// Mitsubishi GX Works2 project: 2023-05-10 #1 생산자동화기능사 1번   PLC: Q03UDV
// 생산자동화기능사

// global labels: Global1
VAR_GLOBAL
  PB1 AT X0 : BOOL;
  PB2 AT X1 : BOOL;
  정지 AT X2 : BOOL;
  공급후진 AT X3 : BOOL;
  공급전진 AT X4 : BOOL;
  가공후진 AT X5 : BOOL;
  가공전진 AT X6 : BOOL;
  송출후진 AT X7 : BOOL;
  송출전진 AT X8 : BOOL;
  배출후진 AT X9 : BOOL;
  배출전진 AT X0A : BOOL;
  매거진 AT X0B : BOOL;
  금속센서 AT X0F : BOOL;
  PB3 AT X0C : BOOL;
  적색 AT Y20 : BOOL;
  황색 AT Y21 : BOOL;
  녹색 AT Y22 : BOOL;
  공급1 AT Y23 : BOOL;
  공급2 AT Y24 : BOOL;
  가공 AT Y25 : BOOL;
  드릴 AT Y26 : BOOL;
  송출 AT Y27 : BOOL;
  배출 AT Y28 : BOOL;
  컨베이어 AT Y29 : BOOL;
  METAL : INT;
END_VAR

PROGRAM 테스트동작
VAR
  STATE : INT;
END_VAR
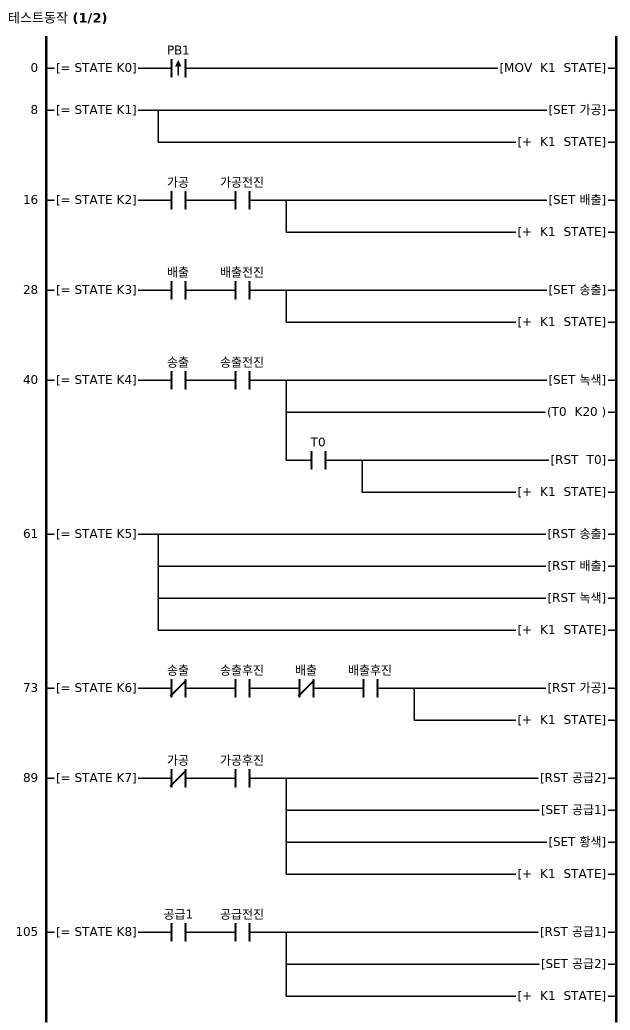
0     LD=     STATE K0
      ANDP    PB1
      MOV     K1 STATE
8     LD=     STATE K1
      SET     가공
      +       K1 STATE
16    LD=     STATE K2
      AND     가공
      AND     가공전진
      SET     배출
      +       K1 STATE
28    LD=     STATE K3
      AND     배출
      AND     배출전진
      SET     송출
      +       K1 STATE
40    LD=     STATE K4
      AND     송출
      AND     송출전진
      SET     녹색
      OUT     T0 K20
      AND     T0
      RST     T0
      +       K1 STATE
61    LD=     STATE K5
      RST     송출
      RST     배출
      RST     녹색
      +       K1 STATE
73    LD=     STATE K6
      ANI     송출
      AND     송출후진
      ANI     배출
      AND     배출후진
      RST     가공
      +       K1 STATE
89    LD=     STATE K7
      ANI     가공
      AND     가공후진
      RST     공급2
      SET     공급1
      SET     황색
      +       K1 STATE
105   LD=     STATE K8
      AND     공급1
      AND     공급전진
      RST     공급1
      SET     공급2
      +       K1 STATE
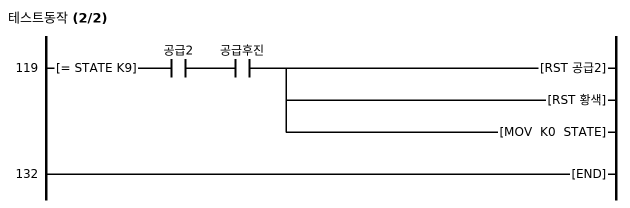
119   LD=     STATE K9
      AND     공급2
      AND     공급후진
      RST     공급2
      RST     황색
      MOV     K0 STATE
132   END
END_PROGRAM

PROGRAM 연속동작
VAR
  COUNT : INT;
  STATE : INT;
  RESET : INT;
END_VAR
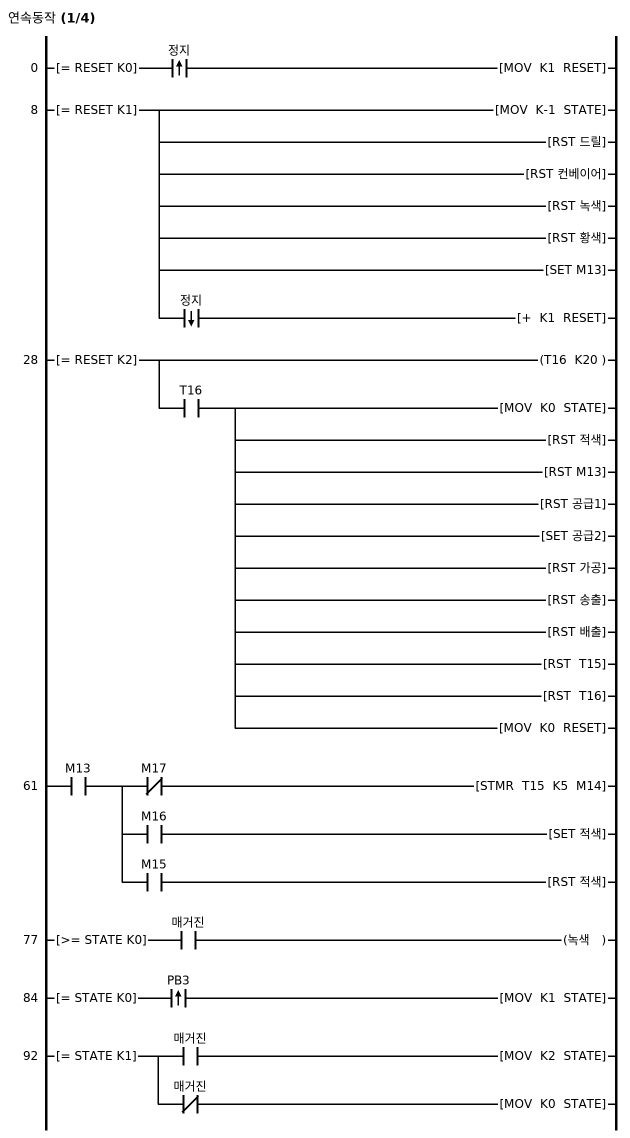
0     LD=     RESET K0
      ANDP    정지
      MOV     K1 RESET
8     LD=     RESET K1
      MOV     K-1 STATE
      RST     드릴
      RST     컨베이어
      RST     녹색
      RST     황색
      SET     M13
      ANDF    정지
      +       K1 RESET
28    LD=     RESET K2
      OUT     T16 K20
      AND     T16
      MOV     K0 STATE
      RST     적색
      RST     M13
      RST     공급1
      SET     공급2
      RST     가공
      RST     송출
      RST     배출
      RST     T15
      RST     T16
      MOV     K0 RESET
61    LD      M13
      MPS
      ANI     M17
      STMR    T15 K5 M14
      MRD
      AND     M16
      SET     적색
      MPP
      AND     M15
      RST     적색
77    LD>=    STATE K0
      AND     매거진
      OUT     녹색
84    LD=     STATE K0
      ANDP    PB3
      MOV     K1 STATE
92    LD=     STATE K1
      MPS
      AND     매거진
      MOV     K2 STATE
      MPP
      ANI     매거진
      MOV     K0 STATE
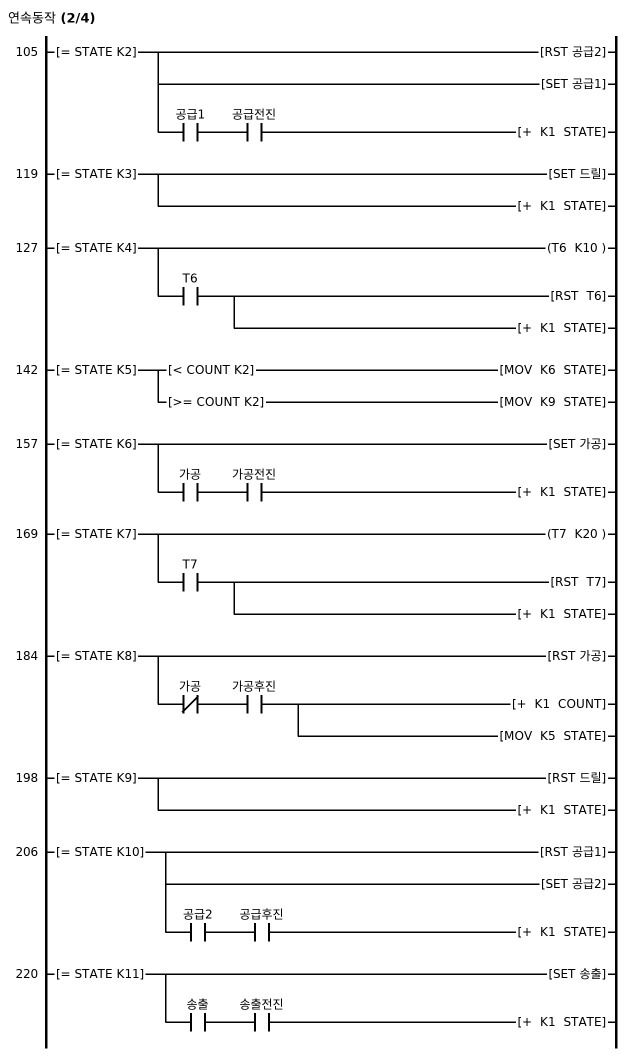
105   LD=     STATE K2
      RST     공급2
      SET     공급1
      AND     공급1
      AND     공급전진
      +       K1 STATE
119   LD=     STATE K3
      SET     드릴
      +       K1 STATE
127   LD=     STATE K4
      OUT     T6 K10
      AND     T6
      RST     T6
      +       K1 STATE
142   LD=     STATE K5
      MPS
      AND<    COUNT K2
      MOV     K6 STATE
      MPP
      AND>=   COUNT K2
      MOV     K9 STATE
157   LD=     STATE K6
      SET     가공
      AND     가공
      AND     가공전진
      +       K1 STATE
169   LD=     STATE K7
      OUT     T7 K20
      AND     T7
      RST     T7
      +       K1 STATE
184   LD=     STATE K8
      RST     가공
      ANI     가공
      AND     가공후진
      +       K1 COUNT
      MOV     K5 STATE
198   LD=     STATE K9
      RST     드릴
      +       K1 STATE
206   LD=     STATE K10
      RST     공급1
      SET     공급2
      AND     공급2
      AND     공급후진
      +       K1 STATE
220   LD=     STATE K11
      SET     송출
      AND     송출
      AND     송출전진
      +       K1 STATE
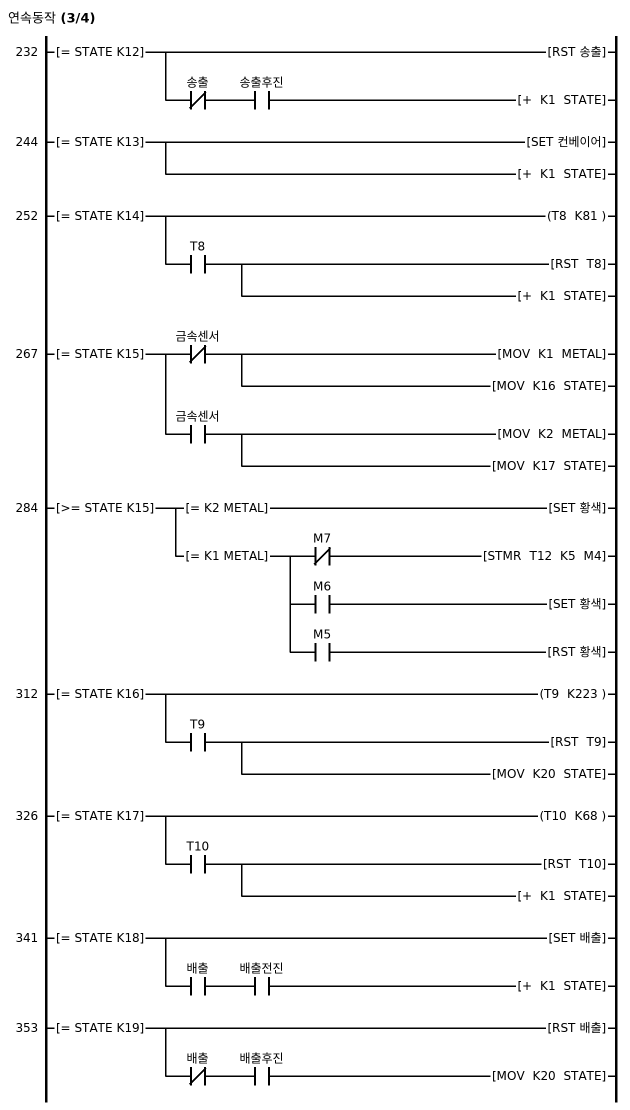
232   LD=     STATE K12
      RST     송출
      ANI     송출
      AND     송출후진
      +       K1 STATE
244   LD=     STATE K13
      SET     컨베이어
      +       K1 STATE
252   LD=     STATE K14
      OUT     T8 K81
      AND     T8
      RST     T8
      +       K1 STATE
267   LD=     STATE K15
      MPS
      ANI     금속센서
      MOV     K1 METAL
      MOV     K16 STATE
      MPP
      AND     금속센서
      MOV     K2 METAL
      MOV     K17 STATE
284   LD>=    STATE K15
      MPS
      AND=    K2 METAL
      SET     황색
      MPP
      AND=    K1 METAL
      MPS
      ANI     M7
      STMR    T12 K5 M4
      MRD
      AND     M6
      SET     황색
      MPP
      AND     M5
      RST     황색
312   LD=     STATE K16
      OUT     T9 K223
      AND     T9
      RST     T9
      MOV     K20 STATE
326   LD=     STATE K17
      OUT     T10 K68
      AND     T10
      RST     T10
      +       K1 STATE
341   LD=     STATE K18
      SET     배출
      AND     배출
      AND     배출전진
      +       K1 STATE
353   LD=     STATE K19
      RST     배출
      ANI     배출
      AND     배출후진
      MOV     K20 STATE
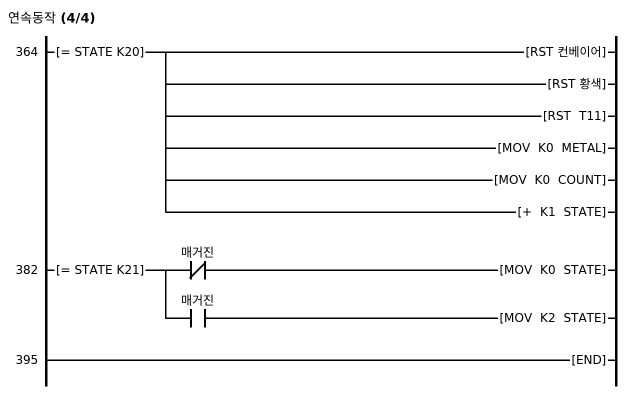
364   LD=     STATE K20
      RST     컨베이어
      RST     황색
      RST     T11
      MOV     K0 METAL
      MOV     K0 COUNT
      +       K1 STATE
382   LD=     STATE K21
      MPS
      ANI     매거진
      MOV     K0 STATE
      MPP
      AND     매거진
      MOV     K2 STATE
395   END
END_PROGRAM

PROGRAM 단속동작
VAR
  STATE : INT;
  RESET : INT;
END_VAR
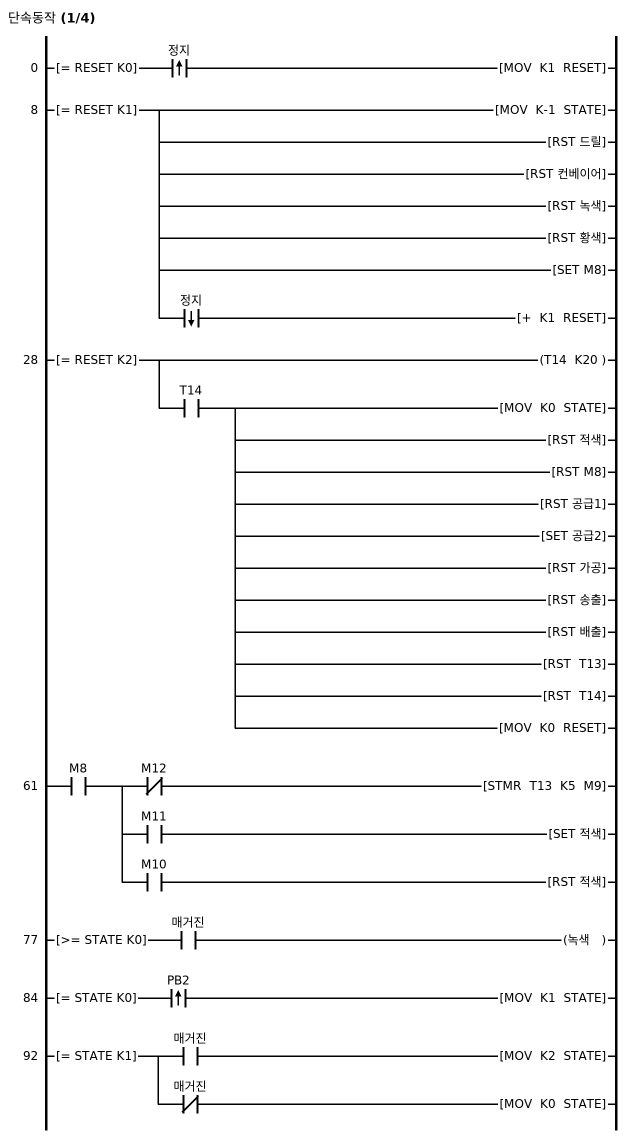
0     LD=     RESET K0
      ANDP    정지
      MOV     K1 RESET
8     LD=     RESET K1
      MOV     K-1 STATE
      RST     드릴
      RST     컨베이어
      RST     녹색
      RST     황색
      SET     M8
      ANDF    정지
      +       K1 RESET
28    LD=     RESET K2
      OUT     T14 K20
      AND     T14
      MOV     K0 STATE
      RST     적색
      RST     M8
      RST     공급1
      SET     공급2
      RST     가공
      RST     송출
      RST     배출
      RST     T13
      RST     T14
      MOV     K0 RESET
61    LD      M8
      MPS
      ANI     M12
      STMR    T13 K5 M9
      MRD
      AND     M11
      SET     적색
      MPP
      AND     M10
      RST     적색
77    LD>=    STATE K0
      AND     매거진
      OUT     녹색
84    LD=     STATE K0
      ANDP    PB2
      MOV     K1 STATE
92    LD=     STATE K1
      MPS
      AND     매거진
      MOV     K2 STATE
      MPP
      ANI     매거진
      MOV     K0 STATE
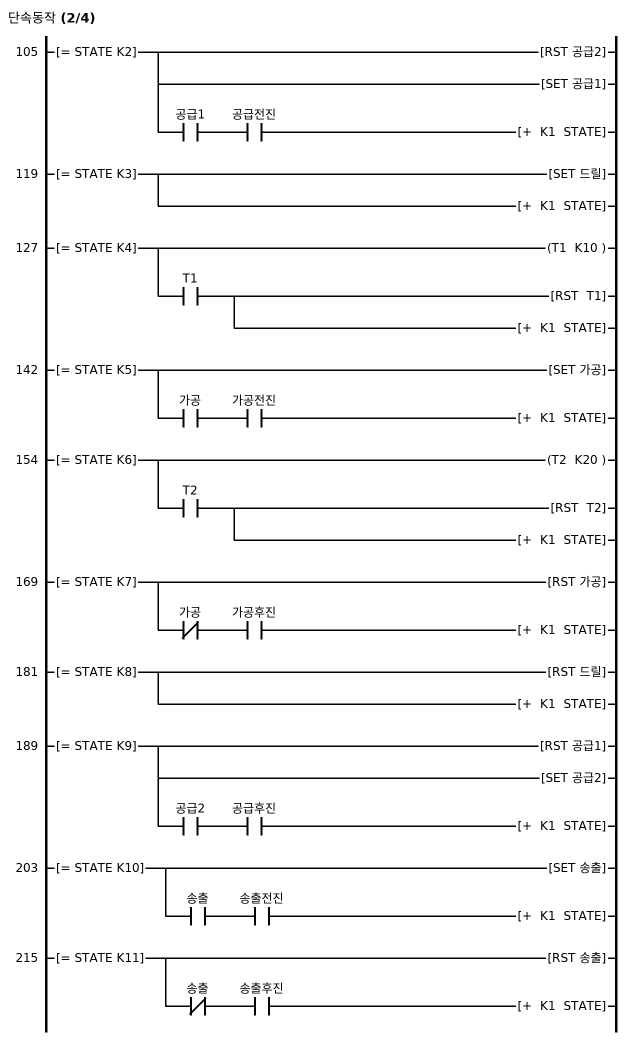
105   LD=     STATE K2
      RST     공급2
      SET     공급1
      AND     공급1
      AND     공급전진
      +       K1 STATE
119   LD=     STATE K3
      SET     드릴
      +       K1 STATE
127   LD=     STATE K4
      OUT     T1 K10
      AND     T1
      RST     T1
      +       K1 STATE
142   LD=     STATE K5
      SET     가공
      AND     가공
      AND     가공전진
      +       K1 STATE
154   LD=     STATE K6
      OUT     T2 K20
      AND     T2
      RST     T2
      +       K1 STATE
169   LD=     STATE K7
      RST     가공
      ANI     가공
      AND     가공후진
      +       K1 STATE
181   LD=     STATE K8
      RST     드릴
      +       K1 STATE
189   LD=     STATE K9
      RST     공급1
      SET     공급2
      AND     공급2
      AND     공급후진
      +       K1 STATE
203   LD=     STATE K10
      SET     송출
      AND     송출
      AND     송출전진
      +       K1 STATE
215   LD=     STATE K11
      RST     송출
      ANI     송출
      AND     송출후진
      +       K1 STATE
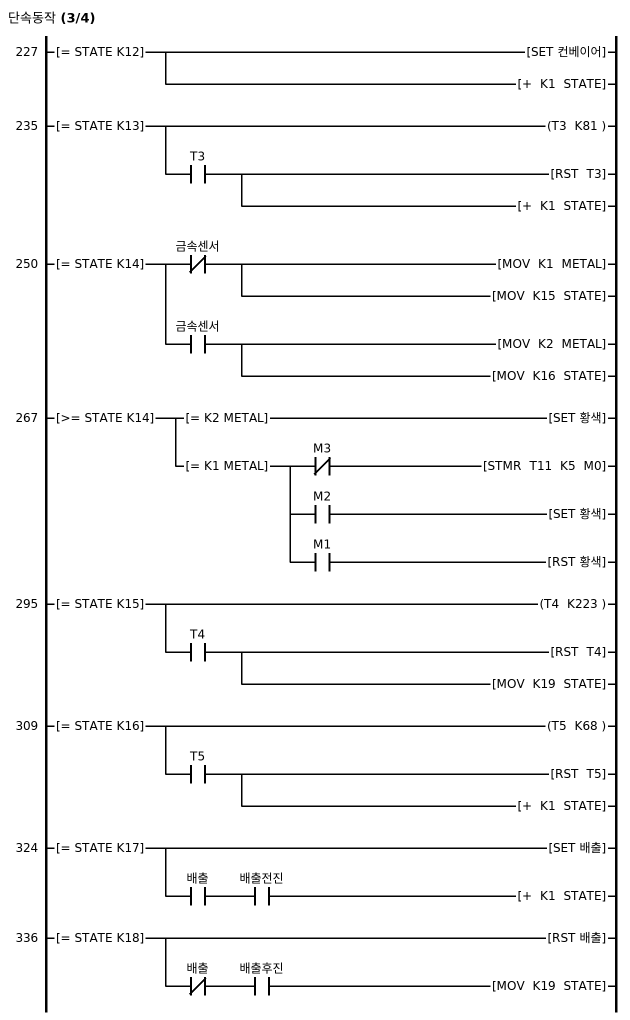
227   LD=     STATE K12
      SET     컨베이어
      +       K1 STATE
235   LD=     STATE K13
      OUT     T3 K81
      AND     T3
      RST     T3
      +       K1 STATE
250   LD=     STATE K14
      MPS
      ANI     금속센서
      MOV     K1 METAL
      MOV     K15 STATE
      MPP
      AND     금속센서
      MOV     K2 METAL
      MOV     K16 STATE
267   LD>=    STATE K14
      MPS
      AND=    K2 METAL
      SET     황색
      MPP
      AND=    K1 METAL
      MPS
      ANI     M3
      STMR    T11 K5 M0
      MRD
      AND     M2
      SET     황색
      MPP
      AND     M1
      RST     황색
295   LD=     STATE K15
      OUT     T4 K223
      AND     T4
      RST     T4
      MOV     K19 STATE
309   LD=     STATE K16
      OUT     T5 K68
      AND     T5
      RST     T5
      +       K1 STATE
324   LD=     STATE K17
      SET     배출
      AND     배출
      AND     배출전진
      +       K1 STATE
336   LD=     STATE K18
      RST     배출
      ANI     배출
      AND     배출후진
      MOV     K19 STATE
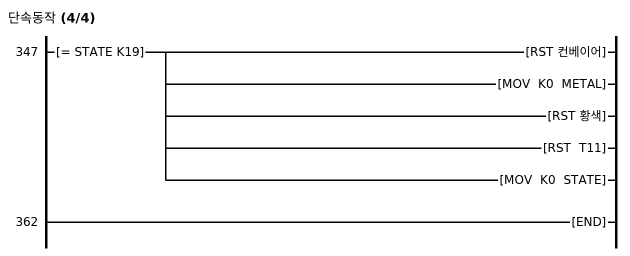
347   LD=     STATE K19
      RST     컨베이어
      MOV     K0 METAL
      RST     황색
      RST     T11
      MOV     K0 STATE
362   END
END_PROGRAM
